(* IEC 61131-3 sources: ICSQuartz/benchmarks/oscat_basic_clean/src, 1 file *)

(* ---- program.st ---- *)
PROGRAM PLC_PRG
VAR_INPUT
    in_in: STRING;
    in_cx: STRING;
END_VAR

CLEAN(in_in, in_cx);

END_PROGRAM
